INTERFACE I_AliasDatatype EXTENDS I_Datatype

PROPERTY PUBLIC BaseType : I_Datatype
GET
END_GET
END_PROPERTY

PROPERTY PUBLIC Identifier : T_MAXSTRING
GET
END_GET
END_PROPERTY

END_INTERFACE

(* stored: Version 1.1.0.1, ProductVersion 3.1.4024.12
   Itf I_AliasDatatype: Id {bec8e99b-9a04-0afe-27d7-e7be6785246b}
   Property BaseType: Id {7c30098c-edb8-0153-0bc1-de3c23a055fd}
   Get Get: Id {328f1f84-e96e-0848-2bfe-08e254da1abe}
   Property Identifier: Id {04cb09dc-7f72-020d-004f-c29896333291}
   Get Get: Id {dac9de76-7974-0110-2888-8c11522082d9} *)
